{attribute 'qualified_only'}
VAR_GLOBAL
		// Event recorder
		fbHistorian	:	HistorianFunctionBlock;

		HistorianDataPacket_EtherCAT	AT	%Q* 	: EthercatDataPacket;
		TransmitApproved				AT	%I*		:	INT;
END_VAR

(* stored: Version 1.1.0.1, ProductVersion 3.1.4022.12
   GVL GVL: Id {72f88768-0d8d-4c67-bbe8-f142f14361b9} *)
